// Implements all three phases and records the order they were called in.

//

// Setup before body, body before teardown, each exactly once. Order is the whole

// contract and nothing else in the library checks it.
FUNCTION_BLOCK OrderedHooksTest IMPLEMENTS I_Test, I_TestSetup, I_TestTeardown
VAR
	_SetupCalls	   : UDINT;
	_BodyCalls	   : UDINT;
	_TeardownCalls : UDINT;

	// Captured at each phase, so the ORDER is provable and not just the counts.
	_BodyAfterSetup	   : BOOL;
	_TeardownAfterBody : BOOL;
	_StatusInTeardown  : E_TestStatus;
END_VAR

PROPERTY BodyAfterSetup : BOOL
GET
BodyAfterSetup := _BodyAfterSetup;
END_GET
END_PROPERTY

PROPERTY BodyCalls : UDINT
GET
BodyCalls := _BodyCalls;
END_GET
END_PROPERTY

METHOD Run : BOOL
VAR_INPUT
	Enable : BOOL;
	Test   : I_TestAssertions;
END_VAR
IF NOT Enable THEN
	Run := TRUE;
	RETURN;
END_IF

_BodyCalls		:= _BodyCalls + 1;
_BodyAfterSetup := (_SetupCalls > 0);
Test.AssertTrue(TRUE, 'body ran');
Run := TRUE;
END_METHOD

METHOD Setup : BOOL
VAR_INPUT
	Enable : BOOL;
	Test   : I_TestAssertions;
END_VAR
_SetupCalls := _SetupCalls + 1;
Setup		:= TRUE;
END_METHOD

PROPERTY SetupCalls : UDINT
GET
SetupCalls := _SetupCalls;
END_GET
END_PROPERTY

// The verdict as teardown saw it. Terminal by then, whatever it is.
PROPERTY StatusInTeardown : E_TestStatus
GET
StatusInTeardown := _StatusInTeardown;
END_GET
END_PROPERTY

METHOD Teardown : BOOL
VAR_INPUT
	Enable : BOOL;
	Test   : I_TestAssertions;
END_VAR
_TeardownCalls	   := _TeardownCalls + 1;
_TeardownAfterBody := (_BodyCalls > 0);

// Readable here on purpose: cleanup may differ by outcome.
_StatusInTeardown := Test.Status;
Teardown		  := TRUE;
END_METHOD

PROPERTY TeardownAfterBody : BOOL
GET
TeardownAfterBody := _TeardownAfterBody;
END_GET
END_PROPERTY

PROPERTY TeardownCalls : UDINT
GET
TeardownCalls := _TeardownCalls;
END_GET
END_PROPERTY

END_FUNCTION_BLOCK

(* stored: Version 1.1.0.1, ProductVersion 3.1.4026.18
   POU OrderedHooksTest: Id {d8a6f79a-7d4f-42c2-ad07-10384effd599}, SpecialFunc None
   Folder I_Test: Id {3a16fa36-1627-4fff-a5b4-5b355e5afd6f}
   Folder I_TestSetup: Id {8cc1caa9-6fac-415c-a4a6-fb7c3a8b135b}
   Folder I_TestTeardown: Id {1d4bdd2f-fe93-4db8-ab28-0615d5b46260}
   Property BodyAfterSetup: Id {490c585b-2a15-4fcf-9084-315d8bdd06c9}
   Get Get: Id {5afc92a3-30ec-42ca-aaae-5c0706c423af}
   Property BodyCalls: Id {d4bb59ac-4f6d-48cd-9869-4db9279e596a}
   Get Get: Id {72b4772e-71ea-47ae-93f9-1c3da6e189e6}
   Method Run: Id {f2fd0ef0-9306-495f-8226-3a744d5a0269}
   Method Setup: Id {8eb8658f-6e18-42f7-b200-5f57fbaf737a}
   Property SetupCalls: Id {00831fdc-68b9-4f49-bada-7829b98ea3e0}
   Get Get: Id {139181bf-7174-4797-b7cc-64ad6e833e93}
   Property StatusInTeardown: Id {da3befda-88d6-4ef0-942c-6b79e927e5d7}
   Get Get: Id {defd2dc2-f868-4250-bb53-b1e73812f200}
   Method Teardown: Id {5701bebb-e08f-41b1-af67-4a7b6fcf8f40}
   Property TeardownAfterBody: Id {abe6133c-193f-41da-afde-76a52ccb0ff9}
   Get Get: Id {20e49ad2-59c5-4ce3-aa31-c97194cb50c0}
   Property TeardownCalls: Id {f1b2c332-b080-47db-b697-e346c3aa9a06}
   Get Get: Id {1a2b19d8-de99-4afc-899a-c3f2aaef26d3} *)
